(* CODESYS project rsCommTcp.library
   Company: ESO
   Description: Library for Tcp communication, e.g. for Lakeshore 336.
      Depends on rsCommCommon.library
   Version: 0.2.0.3
   Placeholder: ESO LDC Comm Tcp Library
   Title: ESO LDC Comm Tcp Library

Project tree, tasks and I/O mapping:
  libraries: ESO LDC Comm Common Library, 0.2.0.3 (ESO); Tc2_Standard, * (Beckhoff Automation GmbH); Tc2_System, * (Beckhoff Automation GmbH); Tc2_TcpIp, * (Beckhoff Automation GmbH); Tc2_Utilities, * (Beckhoff Automation GmbH); Tc3_Module, * (Beckhoff Automation GmbH)
  DUTs/
    Enumerated/
      Comm/
        data type E_TCP_SERVER_STATE
      Devices/
        data type E_TCP_DEVICE_TYPE
    Structures/
      Comm/
        data type T_TCP_SERVER_CTRL
      Devices/
  GVLs/
  lib/
  POUs/
    Comm/
      function block FB_TCP_CLIENT [ST]: M_GetInitialised, M_GetStatus
      function block FB_TCP_SERVER [ST]
    Devices/
      function block FB_LAKESHORE_TCP [ST]: M_Configure, M_GetCommInitialised, M_GetCommStatus, M_UpdateStatus
      function block FB_SIM_TCP_DEVICE_BASE [ST]: M_ActivityDo, M_GenerateRandom_LREAL, M_Get_INT_TO_STRING, M_Get_LREAL_TO_STRING, M_GetRandom_LREAL_TO_STRING, M_GetSimReply
      function block FB_SIM_TCP_LAKESHORE [ST]: M_GetSimReply
    program MAIN [ST]
  VISUs/
    Templates/
      visualisation GUI_TEMPLATE_LAKESHORE_TCP_224
      visualisation GUI_TEMPLATE_LAKESHORE_TCP_336
    visualisation GUI_LAKESHORE_TCP_224
    visualisation GUI_LAKESHORE_TCP_224_SIM
    visualisation GUI_LAKESHORE_TCP_336
    visualisation GUI_LAKESHORE_TCP_336_SIM
  text list GlobalTextList
*)

// DUTs/Enumerated/Comm/E_TCP_SERVER_STATE
{attribute 'qualified_only'}
{attribute 'strict'}
TYPE E_TCP_SERVER_STATE :
(
	NOT_ACCEPTED,
	LISTEN,
	ACCEPT_WAIT,
	RECEIVE_START,
	RECEIVE_WAIT,
	SEND_START,
	SEND_WAIT,
	CLOSE_START,
	CLOSE_WAIT,
	WAIT,
	ERROR
);
END_TYPE

// DUTs/Enumerated/Devices/E_TCP_DEVICE_TYPE
{attribute 'qualified_only'}
{attribute 'strict'}
TYPE E_TCP_DEVICE_TYPE :
(
	LAKESHORE_224 := 0,
	LAKESHORE_336
);
END_TYPE

// DUTs/Structures/Comm/T_TCP_SERVER_CTRL
TYPE T_TCP_SERVER_CTRL :
STRUCT
	(* CTRL *)
	nCommand:		E_RS_COMM_CMD := E_RS_COMM_CMD.NONE;	// Command Number, e.g. SEND
	bExecute:		BOOL;						// Setting to TRUE activates command
	sCmd:			STRING(255) := '';			// Command to be sent
END_STRUCT
END_TYPE

// POUs/Comm/FB_TCP_CLIENT
FUNCTION_BLOCK FB_TCP_CLIENT
VAR_INPUT
	in_bSimulation:		BOOL := FALSE;			// Simulation flag (NOTE: Simulator needed as well)
	in_sDeviceTcpIpAdr: STRING(16);				// Device IP address, e.g. '192.168.0.80' 
	in_nDeviceTcpPort:	UINT;					// Device Tcp port 
	in_sCmdSuffix:		STRING(16) := '$0A';	// Terminator for command, e.g. '$0A' for Lakeshore 336 (LF)
	in_sReplySuffix:	STRING(16) := '$0D$0A';	// Terminator for reply, e.g. '$0D$0A' for Lakeshore 336 (CR/LF) 
	in_nPollingDelay:	DINT := 10;				// Delay after SEND [ms] 
	in_nTimeout:		DINT := 3000;			// Timeout on command reply [ms] 
END_VAR
VAR_OUTPUT
END_VAR
VAR CONSTANT
END_VAR
VAR
	{attribute 'OPC.UA.DA' := '1'}
	cfg:		T_RS_COMM_CFG;				// Config parameters
	{attribute 'OPC.UA.DA' := '1'}
	ctrl:		T_RS_COMM_CTRL;				// Control parameters
	{attribute 'OPC.UA.DA' := '1'}
	{attribute 'OPC.UA.DA.Access' := '1'}
	stat:		T_RS_COMM_STAT;				// Status parameters - ReadOnly

	// Coupler state to be mapped
	i_nCouplerState	AT %I*	: UINT;			(* Link it to Coupler->InfoData->State *)

	fbConnect:		FB_SocketConnect;
	fbSend:			FB_SocketSend;
	fbReceive:		FB_SocketReceive;
	fbClose:		FB_SocketClose;
	
	fbTimer:		TON; // General purpose timer
	fbTimerPoll:	TON; // Receive polling timer

	rxBuffer:		ARRAY[0..1000] OF BYTE;
	sTxFrame:		T_MaxString;


	cmd:			STRING;
	DeviceReply: 	STRING(255);

	State:			INT := E_RS_COMM_STATE.NOT_INIT;
	StateNext:		INT := E_RS_COMM_STATE.IDLE;
	StateNext2:		INT := E_RS_COMM_STATE.IDLE;
	pos:			INT;

	nNumReplies:	DINT := 0;

END_VAR

// Set simulation flag in the status structure
stat.bSimulation	:= in_bSimulation;


(* ============================================
	Check if the HW is OK. 
	The coupler state must be 8, i.e. OPERATIONAL.
============================================== *)
IF i_nCouplerState <> 8  AND  NOT in_bSimulation	THEN	(* If the hardware status is NOT OK, we cannot trust the readings. *)
	stat.nErrorCode	:= E_RS_COMM_ERROR.NOT_IN_OP_STATE;
	stat.sErrorText	:= 'Not in OP state. Is i_nCouplerState linked?';
	stat.nStatus	:= E_RS_COMM_STATUS.ERROR;
	stat.sStatus	:= 'ERROR';
	RETURN;
END_IF

(* ============================================
	Check if Server IP address is given. 
============================================== *)
IF LEN(in_sDeviceTcpIpAdr) = 0 THEN	(* Server IP not set *)
	stat.nErrorCode	:= E_RS_COMM_ERROR.NOT_IN_OP_STATE;
	stat.sErrorText	:= 'Server IP ( var sTcpServerAdr) not set.';
	stat.nStatus	:= E_RS_COMM_STATUS.ERROR;
	stat.sStatus	:= 'ERROR';
	RETURN;
END_IF



(*====================================================
	Handling of commands sent through OPC UA interface.
	Executed only when flag bExecute goes from LOW to HIGH.
	bExecute is reset by the PLC application.
=====================================================*)

IF ctrl.bExecute THEN
	ctrl.bExecute	:= FALSE;
	(* Save last command and reset the command *)
	stat.nLastCommand 	:= ctrl.nCommand;
	ctrl.nCommand		:= E_RS_COMM_CMD.NONE;

	(* Device has to be initialised before being used *)
	IF stat.nLastCommand <> E_RS_COMM_CMD.INIT  AND  NOT stat.bInitialised	THEN
		State 			:= E_RS_COMM_STATE.ERROR;
		stat.nStatus	:= E_RS_COMM_STATUS.ERROR;
		stat.sStatus	:= 'ERROR';
		stat.nErrorCode	:= E_RS_COMM_ERROR.NOT_INIT;
		stat.sErrorText	:= 'Device not initialised.';
		RETURN;
	END_IF

	(* Commands can only be sent when device is IDLE *)
	IF stat.nLastCommand <> E_RS_COMM_CMD.INIT  AND  State <> E_RS_COMM_STATE.IDLE THEN
		State 			:= E_RS_COMM_STATE.ERROR;
		stat.nStatus	:= E_RS_COMM_STATUS.ERROR;
		stat.sStatus	:= 'ERROR';
		stat.nErrorCode	:= E_RS_COMM_ERROR.NOT_IDLE;
		stat.sErrorText	:= 'Device busy. Should be in IDLE to receive commands.';
		RETURN;
	END_IF




	CASE stat.nLastCommand OF
	E_RS_COMM_CMD.INIT:
		stat.bInitialised	:= FALSE;
		stat.sStatus		:= 'INITIALISING';
		stat.nStatus		:= E_RS_COMM_STATUS.BUSY;
		stat.sReply 		:= ''; (* No reply yet *)
		stat.nErrorCode		:= E_RS_COMM_ERROR.OK;
		stat.sErrorText		:= 'OK';
		// Copy input parameters to cfg
		cfg.sCmdSuffix		:= in_sCmdSuffix;
		cfg.sReplySuffix	:= in_sReplySuffix;
		cfg.nTimeout		:= in_nTimeout;

		// Set next state
		State 				:= E_RS_COMM_STATE.RESET;

	E_RS_COMM_CMD.SEND:
		stat.nErrorCode	:= E_RS_COMM_ERROR.OK;
		stat.nStatus	:= E_RS_COMM_STATUS.BUSY;
		stat.sErrorText	:= 'OK';
		stat.sStatus	:= 'BUSY';
		State 			:= E_RS_COMM_STATE.PREPARE_SEND;

	E_RS_COMM_CMD.DISCONNECT:
		stat.nErrorCode		:= E_RS_COMM_ERROR.OK;
		stat.sErrorText		:= 'OK';
		stat.sReply			:= '';
		stat.bInitialised	:= FALSE;

		IF fbConnect.hSocket.handle <> 0  AND  stat.bConnected	THEN
			stat.nStatus	:= E_RS_COMM_STATUS.BUSY;
			stat.sStatus	:= 'DISCONNECTING...';
			fbClose( bExecute:= FALSE );
			fbClose( sSrvNetId := '', hSocket := fbConnect.hSocket, bExecute:= TRUE );
			State	:= E_RS_COMM_STATE.DISCONNECT;
		ELSE
			stat.nStatus	:= E_RS_COMM_STATUS.IDLE;
			stat.sStatus	:= 'IDLE';
			stat.bConnected	:= FALSE;
			State 	:= E_RS_COMM_STATE.NOT_INIT;
		END_IF

	END_CASE

END_IF






(*======================
=======================
 	State machine 
=======================
=======================*)

CASE State OF

E_RS_COMM_STATE.ERROR:
	// Clear buffers
	MEMSET( ADR( sTxFrame ), 0, SIZEOF( sTxFrame ) );
	stat.nStatus	:= E_RS_COMM_STATUS.ERROR;
	stat.sStatus	:= 'ERROR';
//	State 			:= E_RS_COMM_STATE.IDLE;
	RETURN;


E_RS_COMM_STATE.NOT_INIT:
	// Clear buffers
	MEMSET( ADR( sTxFrame ), 0, SIZEOF( sTxFrame ) );
	stat.bInitialised	:= FALSE;
	stat.nErrorCode		:= E_RS_COMM_ERROR.OK;
	stat.sErrorText		:= 'OK';
	stat.nStatus		:= E_RS_COMM_STATUS.NOT_INIT;
	stat.sStatus		:= 'NOT INIT';


E_RS_COMM_STATE.IDLE:
	(* Nothing to do in IDLE *)
	RETURN;


E_RS_COMM_STATE.RESET:
	// Clear buffers
	MEMSET( ADR( sTxFrame ), 0, SIZEOF( sTxFrame ) );
	MEMSET( ADR( rxBuffer ), 0, SIZEOF( rxBuffer ) );
	IF stat.bConnected THEN
		fbClose( bExecute:= FALSE );
		fbClose( sSrvNetId := '', hSocket := fbConnect.hSocket, bExecute:= TRUE );
		StateNext2 	:= E_RS_COMM_STATE.CONNECT;
		State		:= E_RS_COMM_STATE.DISCONNECT;
	ELSE
		fbConnect(	bExecute 	:= FALSE );
		fbConnect(	sSrvNetId 	:= '', 				// Local TCP server
					sRemoteHost := in_sDeviceTcpIpAdr, 
					nRemotePort := in_nDeviceTcpPort,
					tTimeout	:= T#10S, 
					bExecute 	:= TRUE);
		State 	:= E_RS_COMM_STATE.CONNECT;
	END_IF
	
	
E_RS_COMM_STATE.CONNECT:
	fbConnect(	bExecute := FALSE );
	IF fbConnect.bBusy THEN
		RETURN;
	ELSIF fbConnect.bError THEN
		stat.nStatus	:= E_RS_COMM_STATUS.ERROR;
		stat.sStatus	:= 'ERROR';
		stat.nErrorCode	:= E_RS_COMM_ERROR.CONNECT;
		stat.sErrorText	:= 'ERROR. Failed to connect';
		State 			:= E_RS_COMM_STATE.ERROR;
		RETURN;
	ELSE
		stat.nStatus		:= E_RS_COMM_STATUS.IDLE;
		stat.nErrorCode		:= E_RS_COMM_ERROR.OK;
		stat.sErrorText		:= 'OK';
		stat.sStatus		:= 'OK';
		stat.bConnected 	:= TRUE;
		stat.bInitialised	:= TRUE;
		State 				:= E_RS_COMM_STATE.IDLE;
		RETURN;
	END_IF

	

E_RS_COMM_STATE.PREPARE_SEND:
	(*******************************************************************************************
	Here we set the command string, i.e. add suffix if not included in the command.
	Then, the state is changed to  E_RS_COMM_STATE.SEND.
	********************************************************************************************)

	(* Clear the receive buffer *)
	MEMSET( ADR( rxBuffer ), 0, SIZEOF( rxBuffer ) );

	(* Clear reply string *)
	DeviceReply	:= '';

	cmd				:= ctrl.sCmd;

	stat.nStatus	:= E_RS_COMM_STATUS.BUSY;
	stat.sStatus	:= 'BUSY';

	(* Add suffix CR/LF to the user command if missing *)
	pos := FIND(cmd,cfg.sCmdSuffix);
	IF pos = 0 THEN
		cmd := CONCAT(cmd, cfg.sCmdSuffix);
	END_IF

	MEMSET( ADR( sTxFrame ), 0, SIZEOF( sTxFrame ) );
	MEMCPY( ADR( sTxFrame ), ADR( cmd ), INT_TO_UDINT(LEN(cmd)));(* Copy command to send buffer (including the end delimiter) *)

	fbSend( bExecute := FALSE );
	fbSend(	sSrvNetId := '', 
			hSocket	:= fbConnect.hSocket,
			pSrc	:= ADR( sTxFrame ),
			cbLen	:= INT_TO_UDINT(LEN( sTxFrame )),(* String length inclusive the delimiter *)
			tTimeout:= T#2S,
			bExecute:= TRUE );
	
	
	stat.nStatus	:= E_RS_COMM_STATUS.BUSY;
	stat.sStatus	:= 'BUSY';
	nNumReplies		:= 0;		(* Have not received any reply yet. Used for handling multiple replies. *)
	State 			:= E_RS_COMM_STATE.SEND;

	RETURN;


E_RS_COMM_STATE.SEND:
	fbSend( bExecute := FALSE );
	IF fbSend.bBusy THEN
		RETURN;
	ELSIF fbSend.bError  THEN
		// Restart the timer
		fbTimer (IN := FALSE);	// reset timer
		fbTimer (IN := TRUE, PT := DINT_TO_TIME(in_nTimeout));

		stat.nErrorCode	:= E_RS_COMM_ERROR.SEND;
		stat.sErrorText	:= 'Send Failed - Reconnecting...';
		
		stat.bInitialised	:= FALSE;
		stat.nStatus		:= E_RS_COMM_STATUS.ERROR;
		stat.sStatus		:= 'ERROR';

		// Restart socket close
		fbClose( bExecute:= FALSE );
		fbClose( sSrvNetId := '', hSocket := fbConnect.hSocket, bExecute:= TRUE );

		StateNext2 		:= E_RS_COMM_STATE.RESET;
		State 			:= E_RS_COMM_STATE.DISCONNECT;
		
	ELSE
		MEMSET( ADR( rxBuffer ), 0, SIZEOF( rxBuffer ) );	// Clear receive buffer
		stat.sReply := ''; 	// No reply yet 
		(* 	The command has been sent.
			If there is no reply, goto IDLE state.
			Otherwise, goto WAIT_AFTER_SEND state. *)
		fbTimer 	(IN := FALSE);		// reset timer
		fbTimerPoll (IN := FALSE);	// reset timer
		fbTimer		(IN := TRUE, PT := DINT_TO_TIME(in_nTimeout));
		fbTimerPoll	(IN := TRUE, PT := DINT_TO_TIME(in_nPollingDelay));
		State := E_RS_COMM_STATE.WAIT_AFTER_SEND; 	(* Next state is WAIT_AFTER_SEND *)
		RETURN;
	END_IF


E_RS_COMM_STATE.WAIT_AFTER_SEND:
	fbTimerPoll (IN := TRUE);
	IF fbTimerPoll.Q THEN
		fbTimerPoll (IN := FALSE); (* reset timer *)
		IF ctrl.nNumReplies > 0 THEN
			// Start Receive for commands with reply
			fbTimerPoll (IN := TRUE, PT := DINT_TO_TIME(in_nPollingDelay));
			fbReceive(	bExecute := FALSE );
			fbReceive( 	sSrvNetId := '', 
						hSocket	:= fbConnect.hSocket,
						pDest	:= ADR( rxBuffer ),
						cbLen	:= SIZEOF( rxBuffer ),
						bExecute:= TRUE );
	
			State 			:= E_RS_COMM_STATE.RECEIVE;
		ELSE
			(* Prepare next state *)
			State 			:= E_RS_COMM_STATE.IDLE;	 	(* Next state is IDLE *)
			stat.nStatus	:= E_RS_COMM_STATUS.IDLE;
			stat.sStatus	:= 'IDLE';
		END_IF
		RETURN;
	END_IF
	RETURN;

	
E_RS_COMM_STATE.RECEIVE:
	fbReceive( bExecute := FALSE );

	(* Start the timeout timer for receive *)
	fbTimer (IN := TRUE);

	(* Check for timeout. Goto ERROR if timeout expired. *)
	IF fbTimer.Q THEN
		fbTimer (IN := FALSE); (* reset timer *)

		// Restart the timer
		fbTimer (IN := FALSE);	// reset timer
		fbTimer (IN := TRUE, PT := DINT_TO_TIME(in_nTimeout));
		stat.nErrorCode		:= E_RS_COMM_ERROR.TIMEOUT;
		stat.nStatus		:= E_RS_COMM_STATUS.ERROR;
		stat.sErrorText		:= 'Timeout on Receive. Reconnecting...';
		stat.sStatus		:= 'ERROR';
		stat.bInitialised	:= FALSE;

		// Restart socket close. Needed by DISCONNECT
		fbClose( bExecute:= FALSE );
		fbClose( sSrvNetId := '', hSocket := fbConnect.hSocket, bExecute:= TRUE );

		State 			:= E_RS_COMM_STATE.WAIT;			// Wait some time before DISCONNECT
		StateNext		:= E_RS_COMM_STATE.DISCONNECT;	// State after WAIT
		StateNext2		:= E_RS_COMM_STATE.RESET;			// State after DISCONNECT
		RETURN;
	END_IF

	IF fbReceive.bBusy THEN
		RETURN;
	ELSIF fbReceive.bError THEN
		fbTimer (IN := FALSE);	(* reset timer *)

		State 			:= E_RS_COMM_STATE.ERROR;
		stat.nErrorCode	:= E_RS_COMM_ERROR.RECEIVE;
		stat.sErrorText	:= 'Receive Failed';
		RETURN;
	ELSIF fbReceive.nRecBytes > 0 THEN
		(* We have received a reply. Reset timers and triggers. *)
		fbTimer (IN := FALSE); 	(* reset timer *)

		MEMSET( ADR( DeviceReply ), 0, SIZEOF( DeviceReply ) );
		MEMCPY( ADR( DeviceReply ), ADR( rxBuffer ), fbReceive.nRecBytes);(* Copy the received string to the output variable (inclusive the end delimiter) *)

		stat.sReply := DeviceReply;	(* CONCAT the reply *)
		(* Clear the receive buffer ONLY when all replies have been received! *)
		MEMSET( ADR( rxBuffer ), 0, SIZEOF( rxBuffer ) );
		State 			:= E_RS_COMM_STATE.IDLE;
		stat.nStatus	:= E_RS_COMM_STATUS.IDLE;
		stat.sStatus	:= 'IDLE';
		stat.nErrorCode	:= E_RS_COMM_ERROR.OK;
		stat.sErrorText	:= 'OK';
		RETURN;
	ELSE
		// Receive is complete but nothing arrived.
		// Restart Receive.
		fbTimerPoll (IN := FALSE);	// reset timer
		State := E_RS_COMM_STATE.WAIT_AFTER_SEND; 	(* Next state is WAIT_AFTER_SEND *)
		RETURN;
	END_IF



E_RS_COMM_STATE.WAIT:
	// General WAIT state
	// Once the timer expires, go to nextState
	fbTimer (IN := TRUE);
	IF fbTimer.Q THEN
		(* reset timer *)
		fbTimer (IN := FALSE);
		State	:= StateNext;
	END_IF

	
E_RS_COMM_STATE.DISCONNECT:
	fbClose( bExecute:= FALSE );
	// Close any created/opened sockets/connections
	IF fbClose.bBusy THEN
		RETURN;
	ELSIF fbClose.bError THEN
		stat.nStatus	:= E_RS_COMM_STATUS.ERROR;
		stat.sStatus	:= 'ERROR';
		stat.nErrorCode	:= E_RS_COMM_ERROR.DISCONNECT;
		stat.sErrorText	:= 'ERROR. Failed to close connection';
		stat.bConnected	:= FALSE;
		State 			:= E_RS_COMM_STATE.ERROR;
	ELSE
		stat.nStatus	:= E_RS_COMM_STATUS.IDLE;
		stat.sStatus	:= 'IDLE';
		stat.nErrorCode	:= E_RS_COMM_ERROR.OK;
		stat.sErrorText	:= 'OK';
		stat.bConnected	:= FALSE;
		
		IF StateNext2 = E_RS_COMM_STATE.CONNECT	THEN
			// Trigger new connection
			fbConnect(	bExecute 	:= FALSE );
			fbConnect(	sSrvNetId 	:= '', 				// Local TCP server
						sRemoteHost := in_sDeviceTcpIpAdr, 
						nRemotePort := in_nDeviceTcpPort,
						tTimeout	:= T#10S, 
						bExecute 	:= TRUE);
		END_IF
		State 			:= StateNext2;
	END_IF

	

ELSE
(* Unsuported state *)
	State 			:= E_RS_COMM_STATE.ERROR;
	stat.nErrorCode	:= E_RS_COMM_ERROR.WRONG_STATE;
	stat.sErrorText	:= 'Unknown State';
END_CASE



/////////////////////////////////////////////////////////

METHOD M_GetInitialised : BOOL
VAR_INPUT
END_VAR
M_GetInitialised	:= stat.bInitialised;
END_METHOD

METHOD M_GetStatus : E_RS_COMM_STATUS
VAR_INPUT
END_VAR
M_GetStatus	:= stat.nStatus;
END_METHOD

END_FUNCTION_BLOCK

// POUs/Comm/FB_TCP_SERVER
FUNCTION_BLOCK FB_TCP_SERVER
VAR_INPUT
	in_bSimulation:		BOOL := FALSE;			// Simulation flag
	sSrvNetID: 			T_AmsNetID	:= '';		// TwinCAT TCP/IP server network address
	in_sTcpIpAdr: 		STRING(16);				// Server IP address, e.g. '192.168.0.80' 
	in_nTcpPort:		UINT;					// Server Tcp port 
	in_tIdleTime:		TIME	:=  T#10MS;		// Idle time after message received
END_VAR
VAR_OUTPUT
	out_nState: 		E_TCP_SERVER_STATE;
	out_bAccepted: 		BOOL			:= FALSE;(* Accepted connection status *)
	out_bReceived: 		BOOL			:= FALSE;	// Flag if message received
	out_sReceived:		STRING(255)		:= '';		// String received from a client
	bBusy: 			BOOL			:= FALSE;(* BUSY connection status *)
	bError: 		BOOL			:= FALSE;(* ERROR connection status *)
    nErrId: 		DINT			:= 0;		// Error ID
END_VAR
VAR
	{attribute 'OPC.UA.DA' := '1'}
	ctrl:		T_TCP_SERVER_CTRL;				// Control parameters
	{attribute 'OPC.UA.DA' := '1'}
	{attribute 'OPC.UA.DA.Access' := '1'}
	stat:		T_RS_COMM_STAT;				// Status parameters - ReadOnly

	// Coupler state to be mapped
	i_nCouplerState	AT %I*	: UINT;			(* Link it to Coupler->InfoData->State *)

	fbListen	 	: FB_SocketListen;
	fbAccept 		: FB_SocketAccept;
	fbClose			: FB_SocketClose;
	fbReceive		: FB_SocketReceive;
	fbSend			: FB_SocketSend;
	State			: E_TCP_SERVER_STATE;
	StateNext:		E_TCP_SERVER_STATE := E_TCP_SERVER_STATE.NOT_ACCEPTED;		// Next state after Wait
	StateNext2:		E_TCP_SERVER_STATE := E_TCP_SERVER_STATE.NOT_ACCEPTED;		// Exit state from step StateNext

	bDisconnect		: BOOL;(* Disconnect flag, if set the socket will be closed *)

	fbAcceptTimer	: TON;(* Accept poll timer *)
	fbTimer			: TON;(* Receive poll timer *)
	fbRequestTimer	: TON;(* Request timeout timer *)
	
	rxBuffer		: ARRAY[0..1000] OF BYTE;
	sTxFrame		: T_MaxString;
	sRxFrame		: T_MaxString;
	nLenOfString	: UDINT;(* String length inclusive the null delimiter *)
	bEndOfString	: BOOL := FALSE;
	
	sLog:				STRING;
	tPollingTime:	TIME	:= T#100MS;
	
END_VAR

// Set simulation flag in the status structure
stat.bSimulation	:= in_bSimulation;


(* ============================================
	Check if the HW is OK. 
	The coupler state must be 8, i.e. OPERATIONAL.
============================================== *)
IF i_nCouplerState <> 8  AND  NOT in_bSimulation	THEN	(* If the hardware status is NOT OK, we cannot trust the readings. *)
	stat.nErrorCode	:= E_RS_COMM_ERROR.NOT_IN_OP_STATE;
	stat.sErrorText	:= 'Not in OP state. Is i_nCouplerState linked?';
	stat.nStatus	:= E_RS_COMM_STATUS.ERROR;
	stat.sStatus	:= 'ERROR';
	RETURN;
END_IF

(* ============================================
	Check if Server IP address is given. 
============================================== *)
IF LEN(in_sTcpIpAdr) = 0 THEN	(* Server IP not set *)
	stat.nErrorCode	:= E_RS_COMM_ERROR.NOT_IN_OP_STATE;
	stat.sErrorText	:= 'Server IP (in_sTcpIpAdr) not set.';
	stat.nStatus	:= E_RS_COMM_STATUS.ERROR;
	stat.sStatus	:= 'ERROR';
	RETURN;
END_IF



(*====================================================
	Handling of commands sent through OPC UA interface.
	Executed only when flag bExecute goes from LOW to HIGH.
	bExecute is reset by the PLC application.
=====================================================*)

IF ctrl.bExecute THEN
	ctrl.bExecute	:= FALSE;
	(* Save last command and reset the command *)
	stat.nLastCommand 	:= ctrl.nCommand;
	ctrl.nCommand		:= E_RS_COMM_CMD.NONE;

	(* Communication has to be established before being used *)
	IF NOT out_bAccepted	THEN
		stat.nStatus	:= E_RS_COMM_STATUS.ERROR;
		stat.sStatus	:= 'ERROR';
		stat.nErrorCode	:= E_RS_COMM_ERROR.NOT_INIT;
		stat.sErrorText	:= 'Communication not established.';
		RETURN;
	END_IF



	CASE stat.nLastCommand OF

	E_RS_COMM_CMD.SEND:
		stat.nErrorCode	:= E_RS_COMM_ERROR.OK;
		stat.nStatus	:= E_RS_COMM_STATUS.BUSY;
		stat.sErrorText	:= 'OK';
		stat.sStatus	:= 'BUSY';

		// Set command buffer
		MEMSET( ADR( sTxFrame ), 0, SIZEOF( sTxFrame ) );
		MEMCPY( ADR( sTxFrame ), ADR( ctrl.sCmd ), INT_TO_UDINT(LEN(ctrl.sCmd)));

		State 			:= E_TCP_SERVER_STATE.SEND_START;


	END_CASE

END_IF



out_nState	:= State;



CASE State OF
	E_TCP_SERVER_STATE.NOT_ACCEPTED:
		IF fbListen.hListener.handle = 0  OR  fbAccept.nErrId = 32770 THEN
			// Error 32770 means "Socket handle is invalid"
			fbListen(  bExecute := FALSE  );
			fbListen( 	sSrvNetId := sSrvNetID, 
						sLocalHost := in_sTcpIpAdr, 
						nLocalPort := in_nTcpPort, 
						bExecute := TRUE );
						
			State := E_TCP_SERVER_STATE.LISTEN;
		ELSE
			// Trigger connection accept
			fbAccept( bExecute := FALSE );
			fbAccept( sSrvNetId := sSrvNetID, 
						hListener := fbListen.hListener, 
						bExecute:= TRUE );
			fbTimer(IN:=FALSE);
			fbTimer(IN:=TRUE,PT:=T#22S);
			State := E_TCP_SERVER_STATE.ACCEPT_WAIT;
		END_IF
		
		out_bAccepted	:= FALSE;
		out_bReceived	:= FALSE;
		out_sReceived	:= '';
		bBusy		:= TRUE;
		bError		:= FALSE;
		nErrId		:= 0;
		RETURN;

		
	E_TCP_SERVER_STATE.LISTEN:
		fbListen(bExecute:= FALSE );
		IF fbListen.bBusy	THEN
			RETURN;
		ELSIF fbListen.bError AND fbListen.nErrId <> 32771	THEN
			// Error 32771 means that "TcpIp port listener already exists".
			stat.nStatus	:= E_RS_COMM_STATUS.ERROR;
			stat.sStatus	:= 'ERROR';
			stat.nErrorCode	:= E_RS_COMM_ERROR.LISTEN;
			stat.sErrorText	:= 'ERROR. Listen failed. Re-starting...';
			stat.bConnected	:= FALSE;

			out_bAccepted	:= FALSE;
			out_bReceived	:= FALSE;
			out_sReceived	:= '';
			bBusy		:= FALSE;
			bError		:= TRUE;
			nErrId		:= E_RS_COMM_ERROR.LISTEN;
			
			fbTimer(IN:=FALSE);
			fbTimer(IN:=TRUE,PT:=T#10S);
			State 		:= E_TCP_SERVER_STATE.WAIT;			// Goto WAIT
			StateNext	:= E_TCP_SERVER_STATE.NOT_ACCEPTED;	// After WAIT, goto NOT_ACCEPTED
		ELSE
			// Trigger connection accept
			fbAccept( bExecute := FALSE );
			fbAccept( sSrvNetId := sSrvNetID, 
						hListener := fbListen.hListener, 
						bExecute:= TRUE );
			fbTimer(IN:=FALSE);
			fbTimer(IN:=TRUE,PT:=T#2S);
			State := E_TCP_SERVER_STATE.ACCEPT_WAIT;
			RETURN;
		END_IF
	
		
	E_TCP_SERVER_STATE.ACCEPT_WAIT:
		fbAccept( bExecute := FALSE );

		fbTimer(IN:=TRUE);
		IF fbTimer.Q THEN
			// Close the open socket
			sLog	:= 'Closing connection!';
			fbTimer(IN:=FALSE);
			fbTimer(IN:=TRUE,PT:=T#10S);
			fbClose( bExecute := FALSE );
			fbClose( sSrvNetId := sSrvNetID, hSocket:= fbListen.hListener, bExecute:= TRUE );
			State 		:= E_TCP_SERVER_STATE.CLOSE_WAIT;
			RETURN;
		END_IF
		
		IF fbAccept.bBusy THEN
			RETURN;
		ELSIF fbAccept.bError THEN
			stat.nStatus	:= E_RS_COMM_STATUS.ERROR;
			stat.sStatus	:= 'ERROR';
			stat.nErrorCode	:= E_RS_COMM_ERROR.ACCEPT;
			stat.sErrorText	:= 'ERROR. Receive failed';
			stat.bConnected	:= FALSE;
			State 			:= E_TCP_SERVER_STATE.ERROR;
		ELSIF fbAccept.bAccepted THEN
			sLog	:= 'Connection accepted!';
			out_bAccepted	:= TRUE;

			State := E_TCP_SERVER_STATE.RECEIVE_START;
			RETURN;
		ELSE
			// Trigger connection accept
			fbAccept( bExecute := FALSE );
			fbAccept( sSrvNetId := sSrvNetID, 
						hListener := fbListen.hListener, 
						bExecute:= TRUE );
			RETURN;
		END_IF

		
	E_TCP_SERVER_STATE.RECEIVE_START:
	// 25 sec timeout for receive
		fbTimer(IN:=FALSE);
		fbTimer(IN:=TRUE,PT:=T#25S);

		out_bReceived	:= FALSE;
		out_sReceived	:= '';
		bBusy		:= FALSE;
		bError		:= FALSE;
		nErrId		:= 0;
		
		MEMSET( ADR( rxBuffer ), 0, SIZEOF( rxBuffer ) );	// Clear receive buffer
		fbReceive( bExecute := FALSE );
		fbReceive( 	sSrvNetId := sSrvNetID, 
					hSocket	:= fbAccept.hSocket,
					pDest	:= ADR( rxBuffer ),
					cbLen	:= SIZEOF( rxBuffer ),
					bExecute:= TRUE );
					
		State := E_TCP_SERVER_STATE.RECEIVE_WAIT;
		RETURN;



	E_TCP_SERVER_STATE.RECEIVE_WAIT:
		fbReceive(bExecute:= FALSE );

		fbTimer(IN:=TRUE);
		
		IF fbReceive.bBusy	THEN
			RETURN;
		ELSIF fbReceive.bError THEN
			stat.nStatus	:= E_RS_COMM_STATUS.ERROR;
			stat.sStatus	:= 'ERROR';
			stat.nErrorCode	:= E_RS_COMM_ERROR.RECEIVE;
			stat.sErrorText	:= 'ERROR. Receive failed';
			stat.bConnected	:= FALSE;
			State 			:= E_TCP_SERVER_STATE.ERROR;
		ELSIF (fbReceive.nRecBytes > 0) THEN(* Bytes received *)
			sLog		:= 'Received command';
			out_bReceived	:= TRUE;
			bBusy		:= FALSE;
			bError		:= FALSE;
			nErrId		:= 0;

			// Save the received buffer
			MEMSET( ADR( out_sReceived ), 0, SIZEOF( out_sReceived ) );
			MEMCPY( ADR( out_sReceived ), ADR( rxBuffer ), fbReceive.nRecBytes);

			State := E_TCP_SERVER_STATE.RECEIVE_START;
			RETURN;
		ELSIF fbTimer.Q THEN
			// Receive timeout. Close connection and restart.
			State 		:= E_TCP_SERVER_STATE.CLOSE_START;
			RETURN;
		ELSE
			// Nothing received. Trigger Read again.
			fbReceive( 	sSrvNetId := sSrvNetID, 
						hSocket	:= fbAccept.hSocket,
						pDest	:= ADR( rxBuffer ),
						cbLen	:= SIZEOF( rxBuffer ),
						bExecute:= TRUE );
		END_IF
		
		
	E_TCP_SERVER_STATE.SEND_START:
		// Send reply back to the client.
		// sTxFrame is set when we received the command.
		fbSend( bExecute := FALSE );
		fbSend(	sSrvNetId := sSrvNetID, 
				hSocket	:= fbAccept.hSocket,
				pSrc	:= ADR( sTxFrame ),
				cbLen	:= INT_TO_UDINT(LEN( sTxFrame )),// Reply String length 
				bExecute:= TRUE );

		out_bReceived	:= FALSE;
		out_sReceived	:= '';
		bBusy		:= TRUE;
		bError		:= FALSE;
		nErrId		:= 0;
		State 		:= E_TCP_SERVER_STATE.SEND_WAIT;
		RETURN;



	E_TCP_SERVER_STATE.SEND_WAIT:
		fbSend(bExecute:= FALSE );
		IF fbSend.bBusy	THEN
			RETURN;
		ELSIF fbSend.bError THEN
			stat.nStatus	:= E_RS_COMM_STATUS.ERROR;
			stat.sStatus	:= 'ERROR';
			stat.nErrorCode	:= E_RS_COMM_ERROR.SEND;
			stat.sErrorText	:= 'ERROR. Send failed';
			stat.bConnected	:= FALSE;
			State 			:= E_TCP_SERVER_STATE.ERROR;
		ELSE
			sLog	:= 'Reply sent';
			State := E_TCP_SERVER_STATE.RECEIVE_START;
			RETURN;
		END_IF
		
	
	
	E_TCP_SERVER_STATE.CLOSE_START:
		sLog	:= 'Closing connection!';
		fbClose( bExecute := FALSE );
		fbClose( sSrvNetId := sSrvNetID, hSocket:= fbAccept.hSocket, bExecute:= TRUE );
		State := E_TCP_SERVER_STATE.CLOSE_WAIT;

	E_TCP_SERVER_STATE.CLOSE_WAIT:
		fbClose( bExecute := FALSE );
		IF NOT fbClose.bBusy THEN
			out_bAccepted := FALSE;
			IF NOT fbClose.bError THEN
				State := E_TCP_SERVER_STATE.NOT_ACCEPTED;
			ELSE
				sLog	:= 'FB_SocketClose(accepted)';
				State := E_TCP_SERVER_STATE.ERROR;
			END_IF
		END_IF

		
	E_TCP_SERVER_STATE.WAIT:
		fbTimer(IN:=TRUE);
		IF fbTimer.Q	THEN
			State	:= StateNext;
		ELSE
			RETURN;
		END_IF

	
	
	E_TCP_SERVER_STATE.ERROR:
		IF out_bAccepted THEN
			State := E_TCP_SERVER_STATE.CLOSE_START;
		ELSE
			State := E_TCP_SERVER_STATE.NOT_ACCEPTED;
		END_IF

END_CASE

END_FUNCTION_BLOCK

// POUs/Devices/FB_LAKESHORE_TCP
FUNCTION_BLOCK FB_LAKESHORE_TCP EXTENDS FB_LAKESHORE_BASE
VAR_INPUT
	{attribute 'OPC.UA.DA' := '0'}
	in_sDeviceTcpIpAdr: STRING(16);		// Lakeshore IP address, e.g. '192.168.0.80'
	{attribute 'OPC.UA.DA' := '0'}
    in_nDeviceTcpPort:	UINT;			// Lakeshore Tcp port, default 7777 
END_VAR
VAR_OUTPUT
END_VAR
VAR
	{attribute 'OPC.UA.DA' := '0'}
	comm:		FB_TCP_CLIENT;			// Instance of Tcp comm FB. OPC UA Disabled!!!
	
END_VAR


(* Execute comm instance *)
comm(	in_bSimulation		:= in_bSimulation,
		in_sDeviceTcpIpAdr	:= in_sDeviceTcpIpAdr,
		in_nDeviceTcpPort	:= in_nDeviceTcpPort, 
		in_sCmdSuffix		:= in_sCmdSuffix, 
		in_sReplySuffix		:= in_sReplySuffix,
		in_nPollingDelay 	:= 10,
		in_nTimeout			:= 2000);


// Execute the base class object FB_RS_BASE
SUPER^();

METHOD M_Configure
VAR_INPUT
END_VAR
VAR
	// This is OK for models 224 and 336
	cmdList_Init_224:	ARRAY [1..8] OF T_LAKESHORE_COMMAND := [
							(cmd := 'MODE 1', 	nReplies := 0, 	nValues := 0,	offset := 0),
							(cmd := '*IDN?', 	nReplies := 1, 	nValues := 1,	offset := 0),
							(cmd := '', 		nReplies := 0, 	nValues := 0,	offset := 0),
							(cmd := '', 		nReplies := 0, 	nValues := 0,	offset := 0),
							(cmd := '', 		nReplies := 0, 	nValues := 0,	offset := 0),
							(cmd := '', 		nReplies := 0, 	nValues := 0,	offset := 0),
							(cmd := '', 		nReplies := 0, 	nValues := 0,	offset := 0),
							(cmd := '', 		nReplies := 0, 	nValues := 0,	offset := 0)];

	cmdList_Init_336:	ARRAY [1..8] OF T_LAKESHORE_COMMAND := [
							(cmd := 'MODE 1', 	nReplies := 0, 	nValues := 0,	offset := 0),
							(cmd := '*IDN?', 	nReplies := 1, 	nValues := 1,	offset := 0),
							(cmd := '', 		nReplies := 0, 	nValues := 0,	offset := 0),
							(cmd := '', 		nReplies := 0, 	nValues := 0,	offset := 0),
							(cmd := '', 		nReplies := 0, 	nValues := 0,	offset := 0),
							(cmd := '', 		nReplies := 0, 	nValues := 0,	offset := 0),
							(cmd := '', 		nReplies := 0, 	nValues := 0,	offset := 0),
							(cmd := '', 		nReplies := 0, 	nValues := 0,	offset := 0)];


	(*	List of READ commands *)
	(* Lakeshore 218 commands:
		Command "KRDG? 0" requests all 8 temperature values in K.
		Command "CRDG? 0" requests all 8 temperature values in C.
		Reply format: 
			+nn.nnn,+nn.nnn,+nn.nnn,+nn.nnn,+nn.nnn,+nn.nnn,+nn.nnn,+nn.nnn<CR><LF>
	*)

	cmdList_Read_224:	ARRAY [1..16] OF T_LAKESHORE_COMMAND := [
							(cmd := 'KRDG? 0', 	nReplies := 1, 	nValues := 12,	offset := 0),
							(cmd := 'CRDG? 0', 	nReplies := 1, 	nValues := 12,	offset := 12),
							(cmd := '', 		nReplies := 0, 	nValues := 0,	offset := 0),
							(cmd := '', 		nReplies := 0, 	nValues := 0,	offset := 0),
							(cmd := '', 		nReplies := 0, 	nValues := 0,	offset := 0),
							(cmd := '', 		nReplies := 0, 	nValues := 0,	offset := 0),
							(cmd := '', 		nReplies := 0, 	nValues := 0,	offset := 0),
							(cmd := '', 		nReplies := 0, 	nValues := 0,	offset := 0),
							(cmd := '', 		nReplies := 0, 	nValues := 0,	offset := 0),
							(cmd := '', 		nReplies := 0, 	nValues := 0,	offset := 0),
							(cmd := '', 		nReplies := 0, 	nValues := 0,	offset := 0),
							(cmd := '', 		nReplies := 0, 	nValues := 0,	offset := 0),
							(cmd := '', 		nReplies := 0, 	nValues := 0,	offset := 0),
							(cmd := '', 		nReplies := 0, 	nValues := 0,	offset := 0),
							(cmd := '', 		nReplies := 0, 	nValues := 0,	offset := 0),
							(cmd := '', 		nReplies := 0, 	nValues := 0,	offset := 0)];

	cmdList_Read_336:	ARRAY [1..16] OF T_LAKESHORE_COMMAND := [
							(cmd := 'KRDG? A', 	nReplies := 1, 	nValues := 1,	offset := 0),
							(cmd := 'KRDG? B', 	nReplies := 1, 	nValues := 1,	offset := 1),
							(cmd := 'SETP? 1', 	nReplies := 1, 	nValues := 1,	offset := 2),
							(cmd := 'PID? 1', 	nReplies := 1, 	nValues := 3,	offset := 3),
							(cmd := 'RAMP? 1', 	nReplies := 1, 	nValues := 2,	offset := 6),
							(cmd := 'RANGE? 1', nReplies := 1, 	nValues := 1,	offset := 8),
							(cmd := 'HTR? 1', 	nReplies := 1, 	nValues := 1,	offset := 9),
							(cmd := 'SETP? 2', 	nReplies := 1, 	nValues := 1,	offset := 10),
							(cmd := 'PID? 2', 	nReplies := 1, 	nValues := 3,	offset := 11),
							(cmd := 'RAMP? 2', 	nReplies := 1, 	nValues := 2,	offset := 14),
							(cmd := 'RANGE? 2', nReplies := 1, 	nValues := 1,	offset := 16),
							(cmd := 'HTR? 2', 	nReplies := 1, 	nValues := 1,	offset := 17),
							(cmd := 'AOUT? 3', 	nReplies := 1, 	nValues := 1,	offset := 18),
							(cmd := 'AOUT? 4', 	nReplies := 1, 	nValues := 1,	offset := 19),
							(cmd := '', 		nReplies := 0, 	nValues := 0,	offset := 0),
							(cmd := '', 		nReplies := 0, 	nValues := 0,	offset := 0)];

	
END_VAR
// Execute base FB M_Configure().
// This will set cfg.nModel, etc.
SUPER^.M_Configure();

// TODO
// Populate cfg.cmdList_Init and cmdList_Read tables for the specific cfg.nModel.
IF cfg.nModel = 224 THEN
	cfg.cmdList_Init	:= cmdList_Init_224;
	cfg.cmdList_Read	:= cmdList_Read_224;
ELSIF cfg.nModel = 336 THEN
	cfg.cmdList_Init	:= cmdList_Init_336;
	cfg.cmdList_Read	:= cmdList_Read_336;
END_IF


// Set pointers to comm, i.e.
ptrCommCfg	:= ADR(comm.cfg);	(* Pointer to comm.cfg instance *)
ptrCommCtrl	:= ADR(comm.ctrl);	(* Pointer to comm.ctrl instance *)
ptrCommStat	:= ADR(comm.stat);	(* Pointer to comm.stat instance *)

// Set comm suffixes for commands and replies
ptrCommCfg^.sCmdSuffix		:= in_sCmdSuffix;
ptrCommCfg^.sReplySuffix	:= in_sReplySuffix;
END_METHOD

METHOD M_GetCommInitialised : BOOL
VAR_INPUT
END_VAR
M_GetCommInitialised	:= comm.M_GetInitialised();
END_METHOD

METHOD M_GetCommStatus : E_RS_COMM_STATUS
VAR_INPUT
END_VAR
M_GetCommStatus	:= comm.M_GetStatus();
END_METHOD

METHOD M_UpdateStatus
VAR_INPUT
END_VAR
// TODO
//
// Copy values from stat.lrReadings to correspondig stat variables.
// Check M_Configure(). It has to match!
//
// This is an example for model 340.
// This method has to match the list of commands in T_LAKESHORE_CFG::cmdList_Read
IF cfg.nModel = 224 THEN
	// Nothing to do.
	// NOTE: 12 readings [K]: stat.lrArrReadings[0..11].lrValue
	// NOTE: 12 readings [C]: stat.lrArrReadings[12..23].lrValue
	;	
ELSIF cfg.nModel = 336 THEN
	// TODO NOTE: Only loop 1 is handled !!!
	stat.lrKRDG_A		:= stat.lrArrReadings[0].lrValue;
	stat.lrCRDG_A		:= stat.lrKRDG_A - 273.15;
	stat.lrKRDG_B		:= stat.lrArrReadings[1].lrValue;
	stat.lrCRDG_B		:= stat.lrKRDG_B - 273.15;
	// Loop 1
	stat.lrSETP			:= stat.lrArrReadings[2].lrValue;
	stat.nPID_P			:= LREAL_TO_UINT(stat.lrArrReadings[3].lrValue);
	stat.nPID_I			:= LREAL_TO_UINT(stat.lrArrReadings[4].lrValue);
	stat.nPID_D			:= LREAL_TO_UINT(stat.lrArrReadings[5].lrValue);
	stat.bRAMP_On		:= LREAL_TO_BOOL(stat.lrArrReadings[6].lrValue);
	stat.lrRAMP_Rate	:= stat.lrArrReadings[7].lrValue;
	stat.nRANGE			:= LREAL_TO_UINT(stat.lrArrReadings[8].lrValue);
	stat.lrHTR			:= stat.lrArrReadings[9].lrValue;
	// Loop 2
	stat.lrSETP2		:= stat.lrArrReadings[10].lrValue;
	stat.nPID2_P		:= LREAL_TO_UINT(stat.lrArrReadings[11].lrValue);
	stat.nPID2_I		:= LREAL_TO_UINT(stat.lrArrReadings[12].lrValue);
	stat.nPID2_D		:= LREAL_TO_UINT(stat.lrArrReadings[13].lrValue);
	stat.bRAMP2_On		:= LREAL_TO_BOOL(stat.lrArrReadings[14].lrValue);
	stat.lrRAMP2_Rate	:= stat.lrArrReadings[15].lrValue;
	stat.nRANGE2		:= LREAL_TO_UINT(stat.lrArrReadings[16].lrValue);
	stat.lrHTR2			:= stat.lrArrReadings[17].lrValue;
	// Outputs
	stat.lrAOUT3		:= stat.lrArrReadings[18].lrValue;
	stat.lrAOUT4		:= stat.lrArrReadings[19].lrValue;

END_IF
END_METHOD

END_FUNCTION_BLOCK

// POUs/Devices/FB_SIM_TCP_DEVICE_BASE
//
// This is the BASE FB for simulators of TCP based devices.
// This a 
// See also FB_SIM_TCP_LAKESHORE that EXTENDS FB_SIM_TCP_DEVICE_BASE
// 
FUNCTION_BLOCK FB_SIM_TCP_DEVICE_BASE
VAR_INPUT
	// Simulation flag.
	// If TRUE, it means that it doesn't use real network HW but
	// rather localhost IP address '127.0.0.1'.
	// In other words, it simulates a device on the same PLC.
	{attribute 'OPC.UA.DA' := '0'}
	in_bSimulation:		BOOL := FALSE;		
	{attribute 'OPC.UA.DA' := '0'}
	in_bEnable:			BOOL	:= TRUE;	// If TRUE, simulator is active
	{attribute 'OPC.UA.DA' := '0'}
	in_nModel:			DINT;
	{attribute 'OPC.UA.DA' := '0'}
	in_sReplySuffix:	STRING(16);			// Terminator for reply
	{attribute 'OPC.UA.DA' := '0'}
	in_sTcpIpAdr: 		STRING(16);			// Server IP address, e.g. '192.168.0.80' 
	{attribute 'OPC.UA.DA' := '0'}
	in_nTcpPort:		UINT;				// Server Tcp port 
END_VAR
VAR_OUTPUT
END_VAR
VAR
	Device:		FB_TCP_SERVER;
	sReply:		STRING(255);
	ptrDevCtrl:	POINTER TO T_TCP_SERVER_CTRL	:= ADR(Device.ctrl);
END_VAR

IF NOT in_bEnable THEN
	RETURN;
ELSE
	Device(	in_bSimulation	:= in_bSimulation,
			in_sTcpIpAdr	:= in_sTcpIpAdr,
			in_nTcpPort		:= in_nTcpPort);
	
	IF Device.out_bAccepted AND Device.out_bReceived THEN
		// A command has arrived. Send a simulated reply
		sReply	:=	M_GetSimReply(in_sReceived	:=Device.out_sReceived); 
		
		// Trigger SEND
		ptrDevCtrl^.nCommand	:= E_RS_COMM_CMD.SEND;
		ptrDevCtrl^.sCmd		:= sReply;
		ptrDevCtrl^.bExecute	:= TRUE;
	END_IF
END_IF

METHOD M_ActivityDo
VAR_INPUT
END_VAR
END_METHOD

// Get random value in_lrValue + (in_lrNominator * DRAND)
METHOD M_GenerateRandom_LREAL : LREAL
VAR_INPUT
	{attribute 'OPC.UA.DA' := '0'}
	in_lrValue:		LREAL;
	{attribute 'OPC.UA.DA' := '0'}
	in_lrNominator:	LREAL;
END_VAR
VAR
	lrVal:	LREAL;
	lrRand:	LREAL;
	fbDrand:	Tc2_System.DRAND;
END_VAR
VAR_INST
	{attribute 'OPC.UA.DA' := '0'}
	nSeed:	INT := 0;
END_VAR
fbDrand(Seed:=nSeed);
nSeed	:= nSeed + 1;
lrRand	:= in_lrNominator * fbDrand.Num;
lrVal	:= in_lrValue + lrRand;

M_GenerateRandom_LREAL	:= lrVal;
END_METHOD

// Get string with terminator. 
METHOD M_Get_INT_TO_STRING : STRING(255)
VAR_INPUT
	{attribute 'OPC.UA.DA' := '0'}
	in_nValue:		INT;
END_VAR
VAR
END_VAR
// Add sufix, if any
IF in_sReplySuffix <> '' THEN
	M_Get_INT_TO_STRING	:= CONCAT (INT_TO_STRING(in_nValue),in_sReplySuffix);
ELSE
	M_Get_INT_TO_STRING	:= INT_TO_STRING(in_nValue);
END_IF
END_METHOD

// Get string with given precision and add terminator. 
METHOD M_Get_LREAL_TO_STRING : STRING(255)
VAR_INPUT
	{attribute 'OPC.UA.DA' := '0'}
	in_lrValue:		LREAL;
	{attribute 'OPC.UA.DA' := '0'}
	in_nPrecision:	INT	:= 2;	// Number of decimal places, default 2
END_VAR
VAR
	lrVal:		LREAL;
    fbFormat:	FB_FormatString;
	sFormat:	STRING;
    sVal:		T_MaxString;
END_VAR
// Get the input value
lrVal	:= in_lrValue;
// Create a string like '%.2f'
sFormat	:= CONCAT(CONCAT('%.', INT_TO_STRING(in_nPrecision)),'f');
// Print LREAL with <in_nPrecision> decimal places
fbFormat( sFormat := sFormat, arg1 := F_LREAL( lrVal ), sOut => sVal);

// Add sufix, if any
IF in_sReplySuffix <> '' THEN
	M_Get_LREAL_TO_STRING	:= CONCAT (sVal,in_sReplySuffix);
ELSE
	M_Get_LREAL_TO_STRING	:= sVal;
END_IF
END_METHOD

METHOD M_GetRandom_LREAL_TO_STRING : STRING(255)
VAR_INPUT
	{attribute 'OPC.UA.DA' := '0'}
	in_lrValue:		LREAL;
	{attribute 'OPC.UA.DA' := '0'}
	in_lrNominator:	LREAL;
	{attribute 'OPC.UA.DA' := '0'}
	in_nPrecision:	INT	:= 2;	// Number of decimal places, default 2
END_VAR
VAR
	lrVal:		LREAL;
    fbFormat:	FB_FormatString;
	sFormat:	STRING;
    sVal:		T_MaxString;
END_VAR
// Get a random value
lrVal	:= M_GenerateRandom_LREAL(in_lrValue,in_lrNominator);
// Create a string like '%.2f'
sFormat	:= CONCAT(CONCAT('%.', INT_TO_STRING(in_nPrecision)),'f');
// Print LREAL with <in_nPrecision> decimal places
fbFormat( sFormat := sFormat, arg1 := F_LREAL( lrVal ), sOut => sVal);

// Add sufix, if any
IF in_sReplySuffix <> '' THEN
	M_GetRandom_LREAL_TO_STRING	:= CONCAT (sVal,in_sReplySuffix);
ELSE
	M_GetRandom_LREAL_TO_STRING	:= sVal;
END_IF
END_METHOD

METHOD M_GetSimReply : STRING(255)
VAR_INPUT
	{attribute 'OPC.UA.DA' := '0'}
	in_sReceived:	STRING(255);		// String received from a client
END_VAR
VAR
END_VAR
// TODO User: Implement simulater replies in FBs that EXTEND FB_SIM_RS_COMM_BASE.
M_GetSimReply := '';	// Dummy implementation
END_METHOD

END_FUNCTION_BLOCK

// POUs/Devices/FB_SIM_TCP_LAKESHORE
FUNCTION_BLOCK FB_SIM_TCP_LAKESHORE EXTENDS FB_SIM_TCP_DEVICE_BASE
VAR_INPUT
END_VAR
VAR_OUTPUT
END_VAR
VAR
	//
	// Status structure for Lakeshore devices
	//
	bRAMP1_On:		BOOL	:= FALSE;	// RAMP On/Off state
	bRAMP2_On:		BOOL	:= FALSE;	// RAMP On/Off state
	nPID1_P:		UINT	:= 11;		// PID parameter P
	nPID1_I:		UINT	:= 51;		// PID parameter I
	nPID1_D:		UINT	:= 41;		// PID parameter D
	nPID2_P:		UINT	:= 12;		// PID parameter P
	nPID2_I:		UINT	:= 52;		// PID parameter I
	nPID2_D:		UINT	:= 42;		// PID parameter D
	nRANGE1:		UINT	:= 4;		// Heater range
	nRANGE2:		UINT	:= 4;		// Heater range
	lrKRDG_A:		LREAL	:= 283.15;	// Temperature A [K]
	lrKRDG_B:		LREAL	:= 273.15;	// Temperature B [K]
	lrCRDG_A:		LREAL	:= 10.0;	// Temperature A [C]
	lrCRDG_B:		LREAL	:=  0.0;	// Temperature B [C]
	lrRAMP1_Rate:	LREAL	:= 0.0;		// RAMP rate
	lrRAMP2_Rate:	LREAL	:= 0.0;		// RAMP rate
	lrSETP1:		LREAL	:= 283.15;	// Actual Setpoint [K]
	lrSETP1_Target:	LREAL	:= 283.15;	// Target Setpoint [K]
	lrSETP2:		LREAL	:= 282.15;	// Actual Setpoint [K]
	lrSETP2_Target:	LREAL	:= 282.15;	// Target Setpoint [K]
	lrHTR1:			LREAL	:= 0.0;		// Heater output [%]
	lrHTR2:			LREAL	:= 0.0;		// Heater output [%]
	
	fbTimer:		TON;

END_VAR

SUPER^();

METHOD M_GetSimReply : STRING(255)
VAR_INPUT
	{attribute 'OPC.UA.DA' := '0'}
	in_sReceived:	STRING(255);		// String received from a client
END_VAR
VAR
	sReply:	STRING(255);
	lrVal:	LREAL;
	nValue:	UINT;
	i:		INT;
    fbFormat   : FB_FormatString;
    sOut       : T_MaxString;
	nCh:	INT := 8;	// Number of channels for models 218 and 224
END_VAR
IF in_nModel = 336 THEN
	IF FIND (in_sReceived, '*IDN?') > 0 THEN
		M_GetSimReply	:= CONCAT('Lakeshore Simulator',in_sReplySuffix);
	ELSIF FIND (in_sReceived, '*') = 1 THEN
		M_GetSimReply	:= '';	// Ignore commands starting with '*'
	ELSIF FIND (in_sReceived, 'MODE ') > 0 THEN
		M_GetSimReply	:= '';
	ELSIF FIND (in_sReceived, 'CRDG? A') > 0 THEN
		M_GetSimReply	:= M_GetRandom_LREAL_TO_STRING(lrCRDG_A,0.01,2);
	ELSIF FIND (in_sReceived, 'KRDG? A') > 0 THEN
		M_GetSimReply	:= M_GetRandom_LREAL_TO_STRING(lrKRDG_A,0.01,2);
	ELSIF FIND (in_sReceived, 'CRDG? B') > 0 THEN
		M_GetSimReply	:= M_GetRandom_LREAL_TO_STRING(lrCRDG_B,0.01,2);
	ELSIF FIND (in_sReceived, 'KRDG? B') > 0 THEN
		M_GetSimReply	:= M_GetRandom_LREAL_TO_STRING(lrKRDG_B,0.01,2);
	ELSIF FIND (in_sReceived, 'SETP? 1') > 0 THEN
		M_GetSimReply	:= M_Get_LREAL_TO_STRING(lrSETP1_Target,2);
	ELSIF FIND (in_sReceived, 'SETP? 2') > 0 THEN
		M_GetSimReply	:= M_Get_LREAL_TO_STRING(lrSETP2_Target,2);
	ELSIF FIND (in_sReceived, 'PID? 1') > 0 THEN
		fbFormat(	sFormat := '%d,%d,%d', 
					arg1 := F_UINT(nPID1_P), 
					arg2 := F_UINT(nPID1_I), 
					arg3 := F_UINT(nPID1_D), 
					sOut => sOut);
		M_GetSimReply	:= CONCAT(sOut,in_sReplySuffix);
	ELSIF FIND (in_sReceived, 'PID? 2') > 0 THEN
		fbFormat(	sFormat := '%d,%d,%d', 
					arg1 := F_UINT(nPID2_P), 
					arg2 := F_UINT(nPID2_I), 
					arg3 := F_UINT(nPID2_D), 
					sOut => sOut);
		M_GetSimReply	:= CONCAT(sOut,in_sReplySuffix);
	ELSIF FIND (in_sReceived, 'RAMP? 1') > 0 THEN
		nValue	:= BOOL_TO_UINT(bRAMP1_On);	// Convert BOOL to UINT
		fbFormat(	sFormat := '%d,%.2f', 
					arg1 := F_UINT(nValue), 
					arg2 := F_LREAL(lrRAMP1_Rate), 
					sOut => sOut);
		M_GetSimReply	:= CONCAT(sOut,in_sReplySuffix);
	ELSIF FIND (in_sReceived, 'RAMP? 2') > 0 THEN
		nValue	:= BOOL_TO_UINT(bRAMP2_On);	// Convert BOOL to UINT
		fbFormat(	sFormat := '%d,%.2f', 
					arg1 := F_UINT(nValue), 
					arg2 := F_LREAL(lrRAMP2_Rate), 
					sOut => sOut);
		M_GetSimReply	:= CONCAT(sOut,in_sReplySuffix);
	ELSIF FIND (in_sReceived, 'RANGE? 1') > 0 THEN
		M_GetSimReply	:= M_Get_INT_TO_STRING(UINT_TO_INT(nRANGE1));
	ELSIF FIND (in_sReceived, 'RANGE? 2') > 0 THEN
		M_GetSimReply	:= M_Get_INT_TO_STRING(UINT_TO_INT(nRANGE2));
	ELSIF FIND (in_sReceived, 'HTR? 1') > 0 THEN
		M_GetSimReply	:= M_GetRandom_LREAL_TO_STRING(lrHTR1,0.10,2);
	ELSIF FIND (in_sReceived, 'HTR? 2') > 0 THEN
		M_GetSimReply	:= M_GetRandom_LREAL_TO_STRING(lrHTR2,0.10,2);
	ELSIF FIND (in_sReceived, 'AOUT?') > 0 THEN
		M_GetSimReply	:= M_GetRandom_LREAL_TO_STRING(0.0,0.10,2);
	ELSE
		M_GetSimReply	:= CONCAT('777.77',in_sReplySuffix);
	END_IF
ELSIF in_nModel = 224 THEN
	nCh	:= 12;
	
	IF FIND (in_sReceived, 'MODE 1') > 0 THEN
		M_GetSimReply	:= '';
	ELSIF FIND (in_sReceived, '*IDN?') > 0 THEN
		M_GetSimReply	:= CONCAT('Lakeshore Simulator',in_sReplySuffix);
	ELSIF FIND (in_sReceived, 'CRDG?') > 0 THEN
		// Generate a string like:
		// '-233.15,-233.25,-233.35,-233.45,-233.55,-233.65,-233.75,-233.85,-233.95,-233.15,-233.25,-233.35$0D$0A';
		sReply	:= '';
		FOR i:=1 TO nCh DO
			lrVal	:= M_GenerateRandom_LREAL(lrCRDG_A,0.10);
			IF i < nCh THEN
				fbFormat( sFormat := '%+.2f,', arg1 := F_LREAL( lrVal ), sOut => sOut);
			ELSE				
				fbFormat( sFormat := '%+.2f%s', arg1 := F_LREAL( lrVal ), arg2 := F_STRING( in_sReceived ), sOut => sOut);
			END_IF
			sReply	:= CONCAT(sReply, sOut);
		END_FOR
		M_GetSimReply	:= sReply;
	ELSIF FIND (in_sReceived, 'KRDG?') > 0 THEN
		// Generate a string like:
		// '40.15,40.25,40.35,40.45,40.55,40.65,40.75,40.85,40.95,40.15,40.25,40.35$0D$0A';
		sReply	:= '';
		FOR i:=1 TO nCh DO
			lrVal	:= M_GenerateRandom_LREAL(lrKRDG_A,0.10);
			IF i < nCh THEN
				fbFormat( sFormat := '%+.2f,', arg1 := F_LREAL( lrVal ), sOut => sOut);
			ELSE				
				fbFormat( sFormat := '%+.2f%s', arg1 := F_LREAL( lrVal ), arg2 := F_STRING( in_sReceived ), sOut => sOut);
			END_IF
			sReply	:= CONCAT(sReply, sOut);
		END_FOR
		M_GetSimReply	:= sReply;
	ELSE
		M_GetSimReply	:= CONCAT('777.77',in_sReplySuffix);
	END_IF
ELSE
		M_GetSimReply	:= CONCAT('UNKNOWN Lakeshore Model',in_sReplySuffix);
END_IF
END_METHOD

END_FUNCTION_BLOCK

// POUs/MAIN
PROGRAM MAIN
VAR
	// Lakeshore 224 (Ethernet interface)
	{attribute 'OPC.UA.DA' := '1'}
	LS224_TCP:		FB_LAKESHORE_TCP;		// LakeShore based on FB_TCP_CLIENT
	
	// Lakeshore 336 (Ethernet interface)
	{attribute 'OPC.UA.DA' := '1'}
	LS336_TCP:		FB_LAKESHORE_TCP;		// LakeShore based on FB_TCP_CLIENT


	// Lakeshores to be simulated
	{attribute 'OPC.UA.DA' := '1'}
	LS224_TCP_SIM:		FB_LAKESHORE_TCP;		// LakeShore based on FB_TCP_CLIENT
	{attribute 'OPC.UA.DA' := '1'}
	LS336_TCP_SIM:		FB_LAKESHORE_TCP;		// LakeShore based on FB_TCP_CLIENT

	// Simulators
	SIM_LS224_TCP:	FB_SIM_TCP_LAKESHORE;		// LakeShore SIM based on FB_TCP_SERVER
	SIM_LS336_TCP:	FB_SIM_TCP_LAKESHORE;		// LakeShore SIM based on FB_TCP_SERVER


END_VAR


// Lakeshore 224
LS224_TCP(	in_sName			:= 'LS224_TCP',
			in_nModel			:= 224,
			in_nPeriod			:= 1500,
			in_sCmdSuffix		:= '$0D$0A',
			in_sReplySuffix		:= '$0D$0A',
			in_sDeviceTcpIpAdr	:= '192.168.0.12', 
			in_nDeviceTcpPort	:= 7777);

// Lakeshore 336
LS336_TCP(	in_sName			:= 'LS336_TCP',
			in_nModel			:= 336,
			in_nPeriod			:= 1000,
			in_sCmdSuffix		:= '$0A',
			in_sReplySuffix		:= '$0A',
			in_sDeviceTcpIpAdr	:= '192.168.0.80', 
			in_nDeviceTcpPort	:= 7777);

// Dummy Lakeshore 224
// in_bSimulation:= TRUE means that it communicates with a simulator.
// If the simulator is running on the same PLC, in_sDeviceTcpIpAdr:='127.0.0.1'.
// in_nDeviceTcpPort has to match simulator's in_nTcpPort.
// See SIM_LS224_TCP.
LS224_TCP_SIM(
			in_bSimulation		:= TRUE,	
			in_sName			:= 'LS224_TCP_SIM',
			in_nModel			:= 224,
			in_nPeriod			:= 1500,
			in_sCmdSuffix		:= '$0D$0A',
			in_sReplySuffix		:= '$0D$0A',
			in_sDeviceTcpIpAdr	:= '127.0.0.1', 
			in_nDeviceTcpPort	:= 8888);

// Dummy Lakeshore 336
// in_bSimulation:= TRUE means that it communicates with a simulator.
// If the simulator is running on the same PLC, in_sDeviceTcpIpAdr:='127.0.0.1'.
// in_nDeviceTcpPort has to match simulator's in_nTcpPort.
// See SIM_LS336_TCP.
LS336_TCP_SIM(	
			in_bSimulation		:= TRUE,	
			in_sName			:= 'LS336_TCP_SIM',
			in_nModel			:= 336,
			in_nPeriod			:= 1000,
			in_sCmdSuffix		:= '$0A',
			in_sReplySuffix		:= '$0A',
			in_sDeviceTcpIpAdr	:= '127.0.0.1', 
			in_nDeviceTcpPort	:= 7777);


// Lakeshore simulators
SIM_LS224_TCP(	in_bSimulation	:= TRUE,	
				in_bEnable		:= TRUE, 
				in_nModel		:= 224,
				in_sReplySuffix	:= '$0D$0A',
				in_sTcpIpAdr	:= '127.0.0.1',
				in_nTcpPort		:= 8888);

SIM_LS336_TCP(	in_bSimulation	:= TRUE,	
				in_bEnable		:= TRUE, 
				in_nModel		:= 336, 
				in_sReplySuffix	:= '$0A',
				in_sTcpIpAdr	:= '127.0.0.1',
				in_nTcpPort		:= 7777);

END_PROGRAM

// VISUs/Templates/GUI_TEMPLATE_LAKESHORE_TCP_224
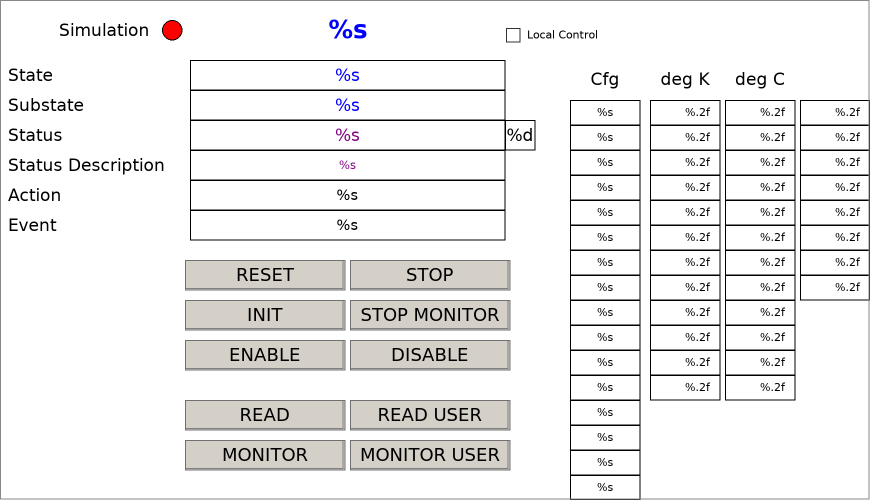
VISUALIZATION GUI_TEMPLATE_LAKESHORE_TCP_224  // 870x500
VAR_IN_OUT
	m_Instance:	FB_LAKESHORE_TCP;
END_VAR
    Rectangle (190,60 315x30), "%s", text variable: m_Instance.stat.sState
    Rectangle (190,90 315x30), "%s", text variable: m_Instance.stat.sSubstate
    Button (185,260 160x30), "RESET", input disabled if: (m_Instance.stat.bLocal = FALSE) <> 0
        OnMouseClick: execute { m_Instance.ctrl.nCommand := E_RS_COMMAND.RESET; m_Instance.ctrl.bExecute := TRUE; }
    Button (185,300 160x30), "INIT", input disabled if: (m_Instance.stat.bLocal = FALSE) <> 0
        OnMouseClick: execute { m_Instance.ctrl.nCommand := E_RS_COMMAND.INIT; m_Instance.ctrl.bExecute := TRUE; }
    Button (350,260 160x30), "STOP", input disabled if: (m_Instance.stat.bLocal = FALSE) <> 0
        OnMouseClick: execute { m_Instance.ctrl.nCommand := E_RS_COMMAND.STOP; m_Instance.ctrl.bExecute := TRUE; }
    Button (185,340 160x30), "ENABLE", input disabled if: (m_Instance.stat.bLocal = FALSE) <> 0
        OnMouseClick: execute { m_Instance.ctrl.nCommand := E_RS_COMMAND.ENABLE; m_Instance.ctrl.bExecute := TRUE; }
    Button (350,340 160x30), "DISABLE", input disabled if: (m_Instance.stat.bLocal = FALSE) <> 0
        OnMouseClick: execute { m_Instance.ctrl.nCommand := E_RS_COMMAND.DISABLE; m_Instance.ctrl.bExecute := TRUE; }
    Rectangle (5,60 180x30), "State"
    Rectangle (5,90 180x30), "Substate"
    Rectangle (190,120 315x30), "%s", text variable: m_Instance.stat.sStatus
    Rectangle (190,150 315x30), "%s", text variable: m_Instance.stat.sErrorText
    Rectangle (5,120 180x30), "Status"
    Rectangle (5,150 180x30), "Status Description"
    Rectangle (190,180 315x30), "%s", text variable: m_Instance.stat.sActionDesc
    Rectangle (190,210 315x30), "%s", text variable: m_Instance.stat.sEventDesc
    Rectangle (5,180 180x30), "Action"
    Rectangle (5,210 180x30), "Event"
    Rectangle (232,12 232x35), "%s", text variable: m_Instance.in_sName
    Rectangle (574,64 62x30), "Cfg"
    Checkbox (504,20 116x30), "Local Control", variable: m_Instance.stat.bLocal
    Rectangle (505,120 30x30), "%d", text variable: m_Instance.stat.nStatus
    Button (185,400 160x30), "READ", tooltip "Single read of all commands in the configuration", input disabled if: (m_Instance.stat.bLocal = FALSE) <> 0
        OnMouseClick: execute { m_Instance.ctrl.nCommand := E_RS_COMMAND.READ; m_Instance.ctrl.bExecute := TRUE; }
    Button (350,400 160x30), "READ USER", tooltip "Single read of user command", input disabled if: (m_Instance.stat.bLocal = FALSE) <> 0
        OnMouseClick: execute { m_Instance.ctrl.nCommand := E_RS_COMMAND.READ_USER; m_Instance.ctrl.bExecute := TRUE; }
    Button (185,440 160x30), "MONITOR", tooltip "Continuously read all commands in the configuration", input disabled if: (m_Instance.stat.bLocal = FALSE) <> 0
        OnMouseClick: execute { m_Instance.ctrl.nCommand := E_RS_COMMAND.MONITOR; m_Instance.ctrl.bExecute := TRUE; }
    Button (350,440 160x30), "MONITOR USER", tooltip "Continuously read the User command", input disabled if: (m_Instance.stat.bLocal = FALSE) <> 0
        OnMouseClick: execute { m_Instance.ctrl.nCommand := E_RS_COMMAND.MONITOR_USER; m_Instance.ctrl.bExecute := TRUE; }
    Rectangle (570,100 70x25), "%s", text variable: m_Instance.cfg.cmdList_Read[1].cmd
    Rectangle (570,125 70x25), "%s", text variable: m_Instance.cfg.cmdList_Read[2].cmd
    Rectangle (570,150 70x25), "%s", text variable: m_Instance.cfg.cmdList_Read[3].cmd
    Rectangle (570,175 70x25), "%s", text variable: m_Instance.cfg.cmdList_Read[4].cmd
    Rectangle (570,200 70x25), "%s", text variable: m_Instance.cfg.cmdList_Read[5].cmd
    Rectangle (570,225 70x25), "%s", text variable: m_Instance.cfg.cmdList_Read[6].cmd
    Rectangle (570,250 70x25), "%s", text variable: m_Instance.cfg.cmdList_Read[7].cmd
    Rectangle (570,275 70x25), "%s", text variable: m_Instance.cfg.cmdList_Read[8].cmd
    Rectangle (570,300 70x25), "%s", text variable: m_Instance.cfg.cmdList_Read[9].cmd
    Rectangle (570,325 70x25), "%s", text variable: m_Instance.cfg.cmdList_Read[10].cmd
    Rectangle (570,350 70x25), "%s", text variable: m_Instance.cfg.cmdList_Read[11].cmd
    Rectangle (570,375 70x25), "%s", text variable: m_Instance.cfg.cmdList_Read[12].cmd
    Rectangle (570,400 70x25), "%s", text variable: m_Instance.cfg.cmdList_Read[13].cmd
    Rectangle (570,425 70x25), "%s", text variable: m_Instance.cfg.cmdList_Read[14].cmd
    Rectangle (570,450 70x25), "%s", text variable: m_Instance.cfg.cmdList_Read[15].cmd
    Rectangle (570,475 70x25), "%s", text variable: m_Instance.cfg.cmdList_Read[16].cmd
    Rectangle (650,100 70x25), "%.2f", text variable: m_Instance.stat.lrArrReadings[0].lrValue
    Rectangle (650,125 70x25), "%.2f", text variable: m_Instance.stat.lrArrReadings[1].lrValue
    Rectangle (650,150 70x25), "%.2f", text variable: m_Instance.stat.lrArrReadings[2].lrValue
    Rectangle (650,175 70x25), "%.2f", text variable: m_Instance.stat.lrArrReadings[3].lrValue
    Rectangle (650,200 70x25), "%.2f", text variable: m_Instance.stat.lrArrReadings[4].lrValue
    Rectangle (650,225 70x25), "%.2f", text variable: m_Instance.stat.lrArrReadings[5].lrValue
    Rectangle (650,250 70x25), "%.2f", text variable: m_Instance.stat.lrArrReadings[6].lrValue
    Rectangle (650,275 70x25), "%.2f", text variable: m_Instance.stat.lrArrReadings[7].lrValue
    Rectangle (650,350 70x25), "%.2f", text variable: m_Instance.stat.lrArrReadings[8].lrValue
    Rectangle (650,375 70x25), "%.2f", text variable: m_Instance.stat.lrArrReadings[9].lrValue
    Rectangle (650,300 70x25), "%.2f", text variable: m_Instance.stat.lrArrReadings[10].lrValue
    Rectangle (650,325 70x25), "%.2f", text variable: m_Instance.stat.lrArrReadings[11].lrValue
    Rectangle (725,100 70x25), "%.2f", text variable: m_Instance.stat.lrArrReadings[12].lrValue
    Rectangle (725,125 70x25), "%.2f", text variable: m_Instance.stat.lrArrReadings[13].lrValue
    Rectangle (725,150 70x25), "%.2f", text variable: m_Instance.stat.lrArrReadings[14].lrValue
    Rectangle (725,175 70x25), "%.2f", text variable: m_Instance.stat.lrArrReadings[15].lrValue
    Rectangle (725,200 70x25), "%.2f", text variable: m_Instance.stat.lrArrReadings[16].lrValue
    Rectangle (725,225 70x25), "%.2f", text variable: m_Instance.stat.lrArrReadings[17].lrValue
    Rectangle (725,250 70x25), "%.2f", text variable: m_Instance.stat.lrArrReadings[18].lrValue
    Rectangle (725,275 70x25), "%.2f", text variable: m_Instance.stat.lrArrReadings[19].lrValue
    Rectangle (654,64 62x30), "deg K"
    Rectangle (729,64 62x30), "deg C"
    Rectangle (725,300 70x25), "%.2f", text variable: m_Instance.stat.lrArrReadings[20].lrValue
    Rectangle (725,325 70x25), "%.2f", text variable: m_Instance.stat.lrArrReadings[21].lrValue
    Rectangle (725,350 70x25), "%.2f", text variable: m_Instance.stat.lrArrReadings[22].lrValue
    Rectangle (725,375 70x25), "%.2f", text variable: m_Instance.stat.lrArrReadings[23].lrValue
    Rectangle (800,100 70x25), "%.2f", text variable: m_Instance.stat.lrArrReadings[24].lrValue
    Rectangle (800,125 70x25), "%.2f", text variable: m_Instance.stat.lrArrReadings[25].lrValue
    Rectangle (800,150 70x25), "%.2f", text variable: m_Instance.stat.lrArrReadings[26].lrValue
    Rectangle (800,175 70x25), "%.2f", text variable: m_Instance.stat.lrArrReadings[27].lrValue
    Rectangle (800,200 70x25), "%.2f", text variable: m_Instance.stat.lrArrReadings[28].lrValue
    Rectangle (800,225 70x25), "%.2f", text variable: m_Instance.stat.lrArrReadings[29].lrValue
    Rectangle (800,250 70x25), "%.2f", text variable: m_Instance.stat.lrArrReadings[30].lrValue
    Rectangle (800,275 70x25), "%.2f", text variable: m_Instance.stat.lrArrReadings[31].lrValue
    Button (350,300 160x30), "STOP MONITOR", tooltip "Stop Monitoring if in OP/MONITORIN state.", input disabled if: (m_Instance.stat.bLocal = FALSE) <> 0
        OnMouseClick: execute { m_Instance.ctrl.nCommand := E_RS_COMMAND.STOPMON; m_Instance.ctrl.bExecute := TRUE; }
    Rectangle (56,15 101x30), "Simulation", invisible if: (m_Instance.stat.bSimulation=FALSE)
    Ellipse (162,20 20x20), tooltip "GREEN=Initialized RED=Not-initialized", text variable: m_Instance.stat.bInitialised, invisible if: (m_Instance.stat.bSimulation=FALSE)
END_VISUALIZATION

// VISUs/Templates/GUI_TEMPLATE_LAKESHORE_TCP_336
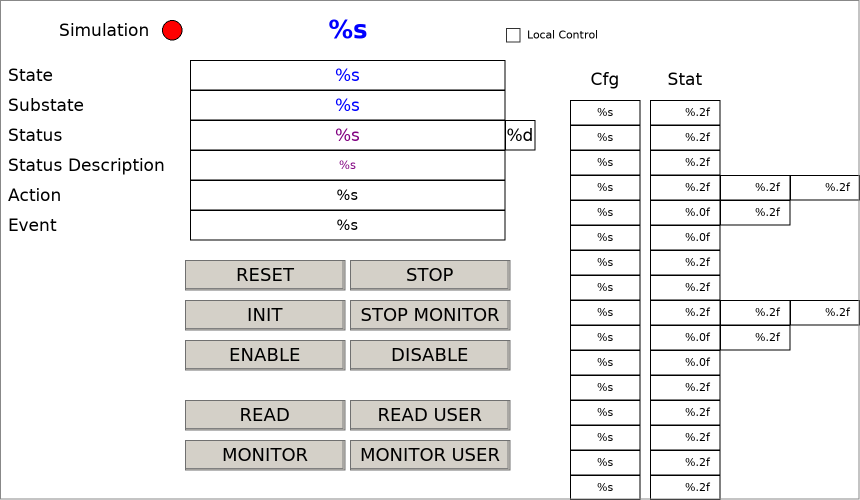
VISUALIZATION GUI_TEMPLATE_LAKESHORE_TCP_336  // 860x500
VAR_IN_OUT
	m_Instance:	FB_LAKESHORE_TCP;
END_VAR
    Rectangle (190,60 315x30), "%s", text variable: m_Instance.stat.sState
    Rectangle (190,90 315x30), "%s", text variable: m_Instance.stat.sSubstate
    Button (185,260 160x30), "RESET", input disabled if: (m_Instance.stat.bLocal = FALSE) <> 0
        OnMouseClick: execute { m_Instance.ctrl.nCommand := E_RS_COMMAND.RESET; m_Instance.ctrl.bExecute := TRUE; }
    Button (185,300 160x30), "INIT", input disabled if: (m_Instance.stat.bLocal = FALSE) <> 0
        OnMouseClick: execute { m_Instance.ctrl.nCommand := E_RS_COMMAND.INIT; m_Instance.ctrl.bExecute := TRUE; }
    Button (350,260 160x30), "STOP", input disabled if: (m_Instance.stat.bLocal = FALSE) <> 0
        OnMouseClick: execute { m_Instance.ctrl.nCommand := E_RS_COMMAND.STOP; m_Instance.ctrl.bExecute := TRUE; }
    Button (185,340 160x30), "ENABLE", input disabled if: (m_Instance.stat.bLocal = FALSE) <> 0
        OnMouseClick: execute { m_Instance.ctrl.nCommand := E_RS_COMMAND.ENABLE; m_Instance.ctrl.bExecute := TRUE; }
    Button (350,340 160x30), "DISABLE", input disabled if: (m_Instance.stat.bLocal = FALSE) <> 0
        OnMouseClick: execute { m_Instance.ctrl.nCommand := E_RS_COMMAND.DISABLE; m_Instance.ctrl.bExecute := TRUE; }
    Rectangle (5,60 180x30), "State"
    Rectangle (5,90 180x30), "Substate"
    Rectangle (190,120 315x30), "%s", text variable: m_Instance.stat.sStatus
    Rectangle (190,150 315x30), "%s", text variable: m_Instance.stat.sErrorText
    Rectangle (5,120 180x30), "Status"
    Rectangle (5,150 180x30), "Status Description"
    Rectangle (190,180 315x30), "%s", text variable: m_Instance.stat.sActionDesc
    Rectangle (190,210 315x30), "%s", text variable: m_Instance.stat.sEventDesc
    Rectangle (5,180 180x30), "Action"
    Rectangle (5,210 180x30), "Event"
    Rectangle (232,12 232x35), "%s", text variable: m_Instance.in_sName
    Rectangle (574,64 62x30), "Cfg"
    Checkbox (504,20 116x30), "Local Control", variable: m_Instance.stat.bLocal
    Rectangle (505,120 30x30), "%d", text variable: m_Instance.stat.nStatus
    Button (185,400 160x30), "READ", tooltip "Single read of all commands in the configuration", input disabled if: (m_Instance.stat.bLocal = FALSE) <> 0
        OnMouseClick: execute { m_Instance.ctrl.nCommand := E_RS_COMMAND.READ; m_Instance.ctrl.bExecute := TRUE; }
    Button (350,400 160x30), "READ USER", tooltip "Single read of user command", input disabled if: (m_Instance.stat.bLocal = FALSE) <> 0
        OnMouseClick: execute { m_Instance.ctrl.nCommand := E_RS_COMMAND.READ_USER; m_Instance.ctrl.bExecute := TRUE; }
    Button (185,440 160x30), "MONITOR", tooltip "Continuously read all commands in the configuration", input disabled if: (m_Instance.stat.bLocal = FALSE) <> 0
        OnMouseClick: execute { m_Instance.ctrl.nCommand := E_RS_COMMAND.MONITOR; m_Instance.ctrl.bExecute := TRUE; }
    Button (350,440 160x30), "MONITOR USER", tooltip "Continuously read the User command", input disabled if: (m_Instance.stat.bLocal = FALSE) <> 0
        OnMouseClick: execute { m_Instance.ctrl.nCommand := E_RS_COMMAND.MONITOR_USER; m_Instance.ctrl.bExecute := TRUE; }
    Rectangle (570,100 70x25), "%s", text variable: m_Instance.cfg.cmdList_Read[1].cmd
    Rectangle (570,125 70x25), "%s", text variable: m_Instance.cfg.cmdList_Read[2].cmd
    Rectangle (570,150 70x25), "%s", text variable: m_Instance.cfg.cmdList_Read[3].cmd
    Rectangle (570,175 70x25), "%s", text variable: m_Instance.cfg.cmdList_Read[4].cmd
    Rectangle (570,200 70x25), "%s", text variable: m_Instance.cfg.cmdList_Read[5].cmd
    Rectangle (570,225 70x25), "%s", text variable: m_Instance.cfg.cmdList_Read[6].cmd
    Rectangle (570,250 70x25), "%s", text variable: m_Instance.cfg.cmdList_Read[7].cmd
    Rectangle (570,275 70x25), "%s", text variable: m_Instance.cfg.cmdList_Read[8].cmd
    Rectangle (570,300 70x25), "%s", text variable: m_Instance.cfg.cmdList_Read[9].cmd
    Rectangle (570,325 70x25), "%s", text variable: m_Instance.cfg.cmdList_Read[10].cmd
    Rectangle (570,350 70x25), "%s", text variable: m_Instance.cfg.cmdList_Read[11].cmd
    Rectangle (570,375 70x25), "%s", text variable: m_Instance.cfg.cmdList_Read[12].cmd
    Rectangle (570,400 70x25), "%s", text variable: m_Instance.cfg.cmdList_Read[13].cmd
    Rectangle (570,425 70x25), "%s", text variable: m_Instance.cfg.cmdList_Read[14].cmd
    Rectangle (570,450 70x25), "%s", text variable: m_Instance.cfg.cmdList_Read[15].cmd
    Rectangle (570,475 70x25), "%s", text variable: m_Instance.cfg.cmdList_Read[16].cmd
    Rectangle (650,100 70x25), "%.2f", text variable: m_Instance.stat.lrArrReadings[0].lrValue
    Rectangle (650,125 70x25), "%.2f", text variable: m_Instance.stat.lrArrReadings[1].lrValue
    Rectangle (650,150 70x25), "%.2f", text variable: m_Instance.stat.lrArrReadings[2].lrValue
    Rectangle (650,175 70x25), "%.2f", text variable: m_Instance.stat.lrArrReadings[3].lrValue
    Rectangle (720,175 70x25), "%.2f", text variable: m_Instance.stat.lrArrReadings[4].lrValue
    Rectangle (790,175 70x25), "%.2f", text variable: m_Instance.stat.lrArrReadings[5].lrValue
    Rectangle (650,200 70x25), "%.0f", text variable: m_Instance.stat.lrArrReadings[6].lrValue
    Rectangle (650,225 70x25), "%.0f", text variable: m_Instance.stat.lrArrReadings[8].lrValue
    Rectangle (650,250 70x25), "%.2f", text variable: m_Instance.stat.lrArrReadings[9].lrValue
    Rectangle (650,275 70x25), "%.2f", text variable: m_Instance.stat.lrArrReadings[10].lrValue
    Rectangle (720,300 70x25), "%.2f", text variable: m_Instance.stat.lrArrReadings[12].lrValue
    Rectangle (790,300 70x25), "%.2f", text variable: m_Instance.stat.lrArrReadings[13].lrValue
    Rectangle (650,300 70x25), "%.2f", text variable: m_Instance.stat.lrArrReadings[11].lrValue
    Rectangle (720,325 70x25), "%.2f", text variable: m_Instance.stat.lrArrReadings[15].lrValue
    Rectangle (650,350 70x25), "%.0f", text variable: m_Instance.stat.lrArrReadings[16].lrValue
    Rectangle (650,375 70x25), "%.2f", text variable: m_Instance.stat.lrArrReadings[17].lrValue
    Rectangle (650,400 70x25), "%.2f", text variable: m_Instance.stat.lrArrReadings[18].lrValue
    Rectangle (650,425 70x25), "%.2f", text variable: m_Instance.stat.lrArrReadings[19].lrValue
    Rectangle (650,450 70x25), "%.2f", text variable: m_Instance.stat.lrArrReadings[20].lrValue
    Rectangle (650,475 70x25), "%.2f", text variable: m_Instance.stat.lrArrReadings[21].lrValue
    Rectangle (654,64 62x30), "Stat"
    Button (350,300 160x30), "STOP MONITOR", tooltip "Stop Monitoring if in OP/MONITORIN state.", input disabled if: (m_Instance.stat.bLocal = FALSE) <> 0
        OnMouseClick: execute { m_Instance.ctrl.nCommand := E_RS_COMMAND.STOPMON; m_Instance.ctrl.bExecute := TRUE; }
    Rectangle (56,15 101x30), "Simulation", invisible if: (m_Instance.stat.bSimulation=FALSE)
    Ellipse (162,20 20x20), tooltip "GREEN=Initialized RED=Not-initialized", text variable: m_Instance.stat.bInitialised, invisible if: (m_Instance.stat.bSimulation=FALSE)
    Rectangle (720,200 70x25), "%.2f", text variable: m_Instance.stat.lrArrReadings[7].lrValue
    Rectangle (650,325 70x25), "%.0f", text variable: m_Instance.stat.lrArrReadings[14].lrValue
END_VISUALIZATION

// VISUs/GUI_LAKESHORE_TCP_224
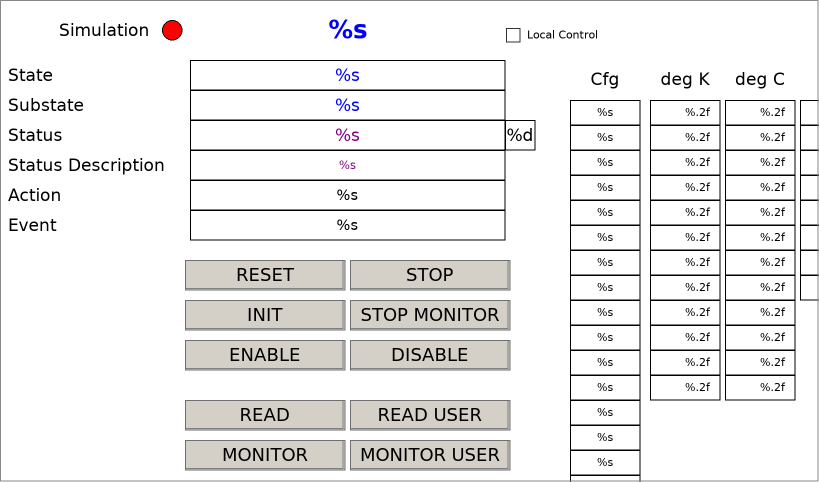
VISUALIZATION GUI_LAKESHORE_TCP_224  // 819x482
    Frame (0,0 817x480)
        shows GUI_TEMPLATE_LAKESHORE_TCP_224(m_Instance := MAIN.LS224_TCP)
END_VISUALIZATION

// VISUs/GUI_LAKESHORE_TCP_224_SIM
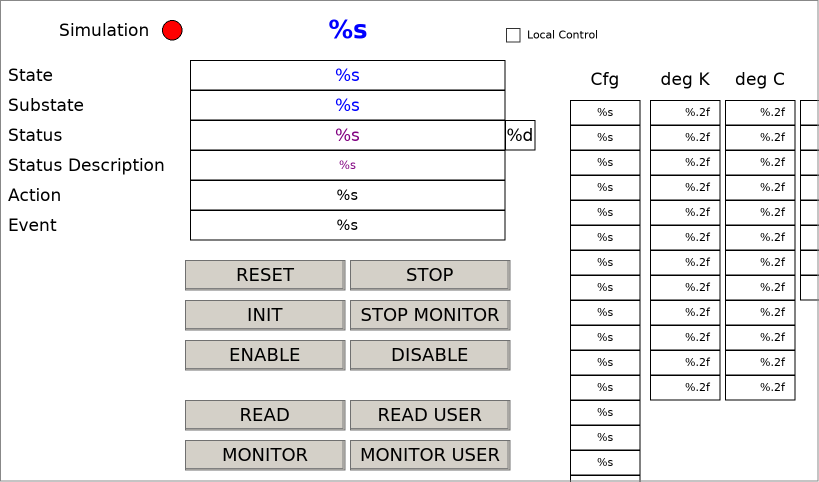
VISUALIZATION GUI_LAKESHORE_TCP_224_SIM  // 819x482
    Frame (0,0 817x480)
        shows GUI_TEMPLATE_LAKESHORE_TCP_224(m_Instance := MAIN.LS224_TCP_SIM)
END_VISUALIZATION

// VISUs/GUI_LAKESHORE_TCP_336
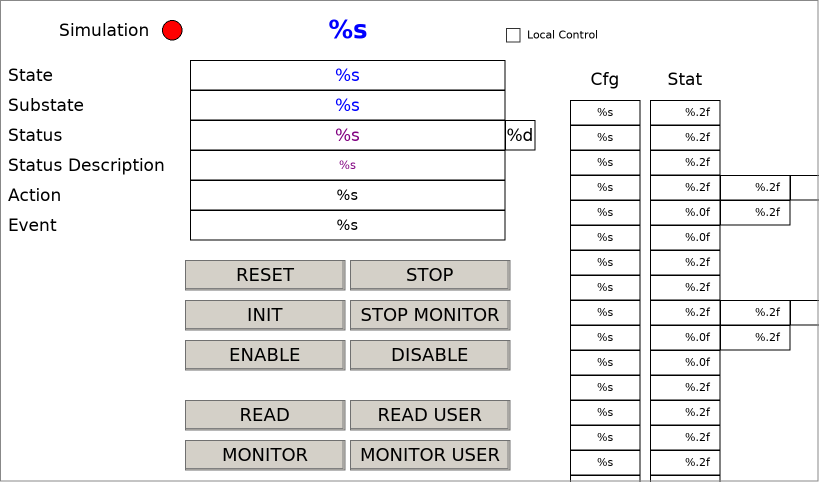
VISUALIZATION GUI_LAKESHORE_TCP_336  // 819x482
    Frame (0,0 817x480)
        shows GUI_TEMPLATE_LAKESHORE_TCP_336(m_Instance := MAIN.LS336_TCP)
END_VISUALIZATION

// VISUs/GUI_LAKESHORE_TCP_336_SIM
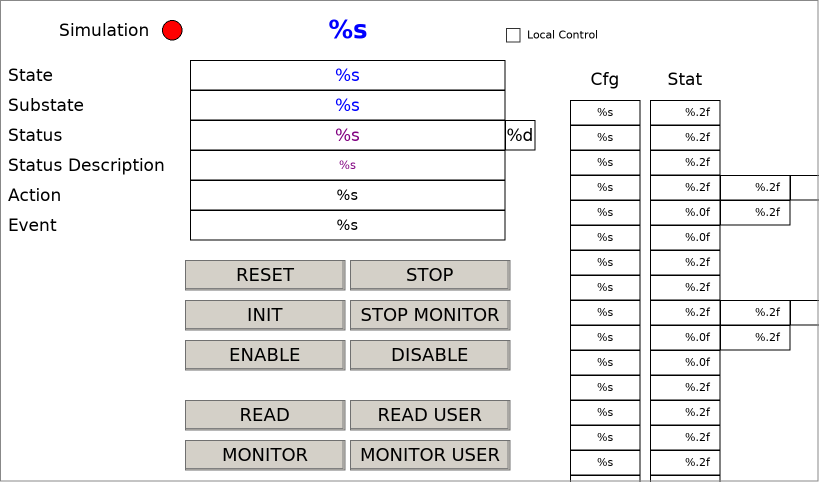
VISUALIZATION GUI_LAKESHORE_TCP_336_SIM  // 819x482
    Frame (0,0 817x480)
        shows GUI_TEMPLATE_LAKESHORE_TCP_336(m_Instance := MAIN.LS336_TCP_SIM)
END_VISUALIZATION
